// TIA Portal V16 export
// export: Created 2025-05-30T16:34:14.9900176Z, ExportSetting WithDefaults, DisplayName Totally Integrated Automation Portal, DisplayVersion V16, DisplayName TIA Portal Version Control Interface, DisplayVersion V16, DisplayName TIA Portal Openness, DisplayVersion V16, DisplayName STEP 7 Professional, DisplayVersion V16, DisplayName STEP 7 Safety, DisplayVersion V16, DisplayName WinCC Advanced, DisplayVersion V16
TYPE "ProductEntry"
// stored: IsFailsafeCompliant false
   STRUCT
      StartTime : Time := T#0ms;
      Active : Bool;
   END_STRUCT;
END_TYPE
